PROGRAM MAIN
VAR
END_VAR

END_PROGRAM

(* stored: Version 1.1.0.1
   POU MAIN: Id {6882f1ea-62e8-4621-88f6-c79ee6b60804} *)
